FUNCTION_BLOCK FB_CoverageFile EXTENDS FB_FileBase


	writeBuffer();

	SUPER^();

END_FUNCTION_BLOCK

(* stored: Version 1.1.0.1, ProductVersion 3.1.4024.13
   POU FB_CoverageFile: Id {73269a4b-8b1b-45f3-8e19-bd0d3a8051c1}, SpecialFunc None *)
